// TwinCAT 3 PLC project PLC
// ProgramVersion: 3.1.4023.0
// libraries:
//   JobManagementFramework, * (Bekchoff Automation K.K.)
//   Tc2_EtherCAT, * (Beckhoff Automation GmbH)
//   Tc2_MC2, * (Beckhoff Automation GmbH)
//   Tc2_Standard, * (Beckhoff Automation GmbH)
//   Tc2_System, * (Beckhoff Automation GmbH)
//   Tc2_Utilities, * (Beckhoff Automation GmbH)
//   Tc3_Module, * (Beckhoff Automation GmbH)
//   VisuSymbols,3.5.10.0,System
// project tree:
//   DUTs/ JobEventReport.TcDUT
//   / GlobalTextList.TcGTLO, PlcTask.TcTTO, Visualization Manager.TcVMO (not stored), VISU_TASK.TcTTO
//   POUs/activities/ FB_Observer.TcPOU, FutureMCGearIn.TcPOU, FutureMCGearInCreator.TcPOU (not stored), FutureMCGearOutCreator.TcPOU (not stored), FutureMCGearOut.TcPOU, FutureMCInching.TcPOU, FutureMCInchingCreator.TcPOU (not stored), FutureMCResetCreator.TcPOU (not stored), FutureMCReset.TcPOU (not stored), FutureMCStopCreator.TcPOU (not stored), FutureMCStop.TcPOU, FutureMCMoveVelocityCreator.TcPOU (not stored), FutureMCMoveVelocity.TcPOU, FutureMCMoveRelativeCreator.TcPOU (not stored), FutureMCMoveRelative.TcPOU, FutureMCMoveAbsolute.TcPOU, FutureMCMoveAbsoluteCreator.TcPOU (not stored), FutureSleepCreator.TcPOU (not stored), FutureMCSetPositionCreator.TcPOU (not stored), FutureMCPower.TcPOU, FutureMCHalt.TcPOU, FutureMCPowerCreator.TcPOU, FutureMCHaltCreator.TcPOU (not stored), FutureMCSetPosition.TcPOU, FutureSleep.TcPOU (not stored)
//   POUs/ MAIN.TcPOU
//   VISUs/ Visualization.TcVIS
// real-time tasks:
//   TASK PlcTask: cycle T#1ms, priority 4, ADS port 350
//   TASK VISU_TASK1: cycle T#50000us, priority 30, ADS port 352
// motion (NC):
//   TASK NC-Task 1 SAF: cycle T#2ms, priority 6, ADS port 501
//   TASK NC-Task 1 SVB: cycle T#10ms, priority 10, ADS port 511
//   AXIS Axis 1 (id 1)
//     General: UnitName=Degree
//     Dynamic: AccelerationMaximum=29071, DecelerationMaximum=29071, Acceleration=14535, Deceleration=14535, Jerk=43605
//     Velo: RefSearch=96.9, RefSync=96.9, SlowManual=484.5, FastManual=2907, Fast=9690, Maximum=9690
//     OtherSettings: AllowMotionCmdToSlave=true
//     encoder EncType=19
//       EncPara: ScaleFactorNumerator=360, ScaleFactorDenominator=1048576, MaxCount=#xffffffff
//     drive DrvType=16
//       DrvPara: MaxCount=#xffffffff, DriveControlDWord=#x00020100
//         Analog: VeloReferenz=10659, VeloScale=32, TorqueSetpointScale=10, ScaleFactorActTorque=0.1
//         TimeComp: TaskDelayCycles=1
//     controller CtrType=1
//       CtrPara: PriorControlFactor=1
//         Observer: BandWidth=20
//   AXIS Axis 2 (id 2)
//     General: UnitName=Degree
//     Dynamic: AccelerationMaximum=29071, DecelerationMaximum=29071, Acceleration=14535, Deceleration=14535, Jerk=43605
//     Velo: RefSearch=96.9, RefSync=96.9, FastManual=200, Fast=9690, Maximum=9690
//     OtherSettings: AllowMotionCmdToSlave=true, PulseDistancePos=1, PulseDistanceNeg=1
//     encoder EncType=19
//       EncPara: ScaleFactorNumerator=360, ScaleFactorDenominator=1048576, Inverse=true, MaxCount=#xffffffff
//     drive DrvType=16
//       DrvPara: Inverse=true, MaxCount=#xffffffff, DriveControlDWord=#x00020100
//         Analog: VeloReferenz=10659, VeloScale=32, TorqueSetpointScale=10, ScaleFactorActTorque=0.1
//         TimeComp: TaskDelayCycles=1
//     controller CtrType=1
//       CtrPara: PriorControlFactor=1
//         Observer: BandWidth=20
// I/O:
//   DEVICE Device 2 (EtherCAT), AmsNetId 169.254.89.239.3.1
//     Term 1 (EK1101) [EK1101 EtherCAT Coupler (2A E-Bus, ID switch)]
//       Drive 2 (EL7201-0011) [EL7201-0011 1Ch. DS402 Servo motor output stage with OCT (50V, 4A)]
//       Drive 3 (EL7201-0011) [EL7201-0011 1Ch. DS402 Servo motor output stage with OCT (50V, 2.8A RMS)]
//       Term 4 (EL9011) [EL9011 End Terminal]
// variable links:
//   NC-Task 1 SAF/Axes/Axis 1 <-> Device 2 (EtherCAT)/Term 1 (EK1101)/Drive 2 (EL7201-0011)
//     Drive/Inputs/In/nDataIn1 <-> DS402 Following error actual value/Following error actual value
//     Drive/Inputs/In/nDcOutputTime <-> InfoData/DcOutputShift
//     Drive/Inputs/In/nState1 <-> DS402 Statusword/Statusword
//     Drive/Inputs/In/nState2 <-> DS402 Statusword/Statusword @bit 8
//     Drive/Inputs/In/nState4 @bit 1 <-> WcState/InputToggle
//     Drive/Inputs/In/nState4 <-> WcState/WcState
//     Drive/Outputs/Out/nCtrl1 <-> DS402 Controlword/Controlword
//     Drive/Outputs/Out/nCtrl2 <-> DS402 Controlword/Controlword @bit 8
//     Drive/Outputs/Out/nDataOut1 <-> DS402 Target position/Target position
//     Enc/Inputs/In/nDataIn1 <-> DS402 Position actual value/Position actual value
//     Enc/Inputs/In/nDcInputTime <-> InfoData/DcInputShift
//     Enc/Inputs/In/nState4 @bit 1 <-> WcState/InputToggle
//     Enc/Inputs/In/nState4 <-> WcState/WcState
//   NC-Task 1 SAF/Axes/Axis 2 <-> Device 2 (EtherCAT)/Term 1 (EK1101)/Drive 3 (EL7201-0011)
//     Drive/Inputs/In/nDataIn1 <-> DS402 Following error actual value/Following error actual value
//     Drive/Inputs/In/nDcOutputTime <-> InfoData/DcOutputShift
//     Drive/Inputs/In/nState1 <-> DS402 Statusword/Statusword
//     Drive/Inputs/In/nState2 <-> DS402 Statusword/Statusword @bit 8
//     Drive/Inputs/In/nState4 @bit 1 <-> WcState/InputToggle
//     Drive/Inputs/In/nState4 <-> WcState/WcState
//     Drive/Outputs/Out/nCtrl1 <-> DS402 Controlword/Controlword
//     Drive/Outputs/Out/nCtrl2 <-> DS402 Controlword/Controlword @bit 8
//     Drive/Outputs/Out/nDataOut1 <-> DS402 Target position/Target position
//     Enc/Inputs/In/nDataIn1 <-> DS402 Position actual value/Position actual value
//     Enc/Inputs/In/nDcInputTime <-> InfoData/DcInputShift
//     Enc/Inputs/In/nState4 @bit 1 <-> WcState/InputToggle
//     Enc/Inputs/In/nState4 <-> WcState/WcState
//   PLC/PLC Instance <-> NC-Task 1 SAF/Axes/Axis 1
//     PlcTask Inputs/MAIN.stAxis1.NcToPlc <-> Outputs/ToPlc
//     PlcTask Outputs/MAIN.stAxis1.PlcToNc <-> Inputs/FromPlc
//   PLC/PLC Instance <-> NC-Task 1 SAF/Axes/Axis 2
//     PlcTask Inputs/MAIN.stAxis2.NcToPlc <-> Outputs/ToPlc
//     PlcTask Outputs/MAIN.stAxis2.PlcToNc <-> Inputs/FromPlc

CONFIGURATION PLC
    RESOURCE PLC ON TwinCAT3
        TASK PlcTask(INTERVAL := T#1ms, PRIORITY := 4);
        TASK VISU_TASK(INTERVAL := T#50000us, PRIORITY := 30);
        PROGRAM MAIN WITH PlcTask : MAIN;
        PROGRAM VisuElems_Visu_Prg WITH VISU_TASK : VisuElems.Visu_Prg;
    END_RESOURCE
END_CONFIGURATION

// ---- DUTs/JobEventReport.TcDUT
{attribute 'pack_mode' := '1'}
TYPE JobEventReport :
STRUCT
	{attribute 'TcAnalytics'}
	subject	: STRING(256);
	 {attribute 'TcAnalytics'}
	job_id	: STRING(256);
	 {attribute 'TcAnalytics'}
	old_state	: STRING(16);
	 {attribute 'TcAnalytics'}
	new_state	: STRING(16);
	 {attribute 'TcAnalytics'}
	record_time	: jobmgmt.T_FILETIME64;
END_STRUCT
END_TYPE

// ---- POUs/MAIN.TcPOU
PROGRAM MAIN
VAR
	work_number	: ULINT;
	act_dc_time : T_DCTIME64;
	dc_task_time : T_DCTIME64;
	dc_tick_time : T_DCTIME64;
	diff_time : T_DCTIME64;
	fbConvertDcTimeToPos : ConvertDcTimeToPos;
	position_at_task_start_point : LREAL;
	position_diff : LREAL;
	dc_time_array : ARRAY [0..1] OF T_DCTIME32;

	fbPower1:mc_power;
	fbPower2:mc_power;
	fbJog:MC_Jog;
	basic_job : FB_Executor;
	demo_job : FB_Executor;
	gear_in_job : FB_Executor;
	init_pos_job : FB_Executor;
	jog_plus_job : FB_Executor;
	jog_minus_job : FB_Executor;
	fb_observer : FB_Observer;
	job_reset : BOOL;
	
	mc_power_future_creator: FutureMCPowerCreator;
	mc_reset_future_creator: FutureMCResetCreator;
	mc_set_position_future_creator: FutureMCSetPositionCreator;
	mc_inching_future_creator : FutureMCInchingCreator;
	mc_gear_in_future_creator : FutureMCGearInCreator;
	mc_gear_out_future_creator : FutureMCGearOutCreator;
	mc_move_rel_future_creator : FutureMCMoveRelativeCreator;
	mc_move_abs_future_creator : FutureMCMoveAbsoluteCreator;
	mc_move_velocity_future_creator: FutureMCMoveVelocityCreator;
	mc_stop_future_creator: FutureMCStopCreator;
	sleep_creator : FutureSleepCreator;

	
	iState:INT;
	stAxis1:axis_ref;
	stAxis2:axis_ref;
	bStart: BOOL;
	bJogPlus: BOOL;
	bJogMinus: BOOL;
	bPower: BOOL;
	_bPower : BOOL;
	iPowerState : UINT;
	bReset:BOOL;
	bError:BOOL;
	bAllAxisPowerOn: BOOL;
	bInsync:BOOL;
	create_container: INT;
	boot_up : BOOL := TRUE;
	i: UINT;
	
	quit: INT;
END_VAR


act_dc_time := F_GetActualDcTime64();
dc_task_time := F_GetCurDcTaskTime64();
dc_tick_time := F_GetCurDcTickTime64();

MEMCPY(ADR(dc_time_array), ADR(dc_task_time), SIZEOF(dc_task_time));

fbConvertDcTimeToPos(nAxisId := 1, nSubIdx := 16#10000, dcTime := dc_time_array[0] + 300000);
position_at_task_start_point := fbConvertDcTimeToPos.fPosition;
position_diff := stAxis1.NcToPlc.ActPos - fbConvertDcTimeToPos.fPosition;

diff_time := act_dc_time - dc_task_time;

IF boot_up THEN
	basic_job.create_container(ContainerType.PARALLEL_QUEUE, 'BASIC');
	basic_job.continuous_mode := TRUE;
	basic_job.id := 'M1';
	basic_job.job_event_reporter := fb_observer;
	JobCreate_PosInit(init_pos_job);
	JobCreate_GearIn(gear_in_job);
	JobCreateDemo(demo_job);
	
	

	mc_inching_future_creator.set_parameters(stAxis2, TRUE,1 , 100);
	jog_plus_job.create_future(mc_inching_future_creator,'JOG_PLUS');
	
	mc_inching_future_creator.set_parameters(stAxis2, FALSE, 1, 100);		
	jog_minus_job.create_future(mc_inching_future_creator,'JOG_MINUS');

	boot_up := FALSE;
END_IF


fbPower1(Axis := stAxis1, Enable := bPower, Enable_Positive := TRUE, Enable_Negative := TRUE, Override := 100.0);
fbPower2(Axis := stAxis2, Enable := bPower, Enable_Positive := TRUE, Enable_Negative := TRUE, Override := 100.0);

(*
IF NOT fbPower1.Status AND NOT fbPower2.Status THEN
	IF demo_job.reset(FALSE) THEN
		iState := 0;
	END_IF
END_IF
*)

CASE iState OF
	0:
		IF fbPower1.Status AND fbPower2.Status THEN
			IF init_pos_job.init() THEN
				basic_job.children.append_job(init_pos_job);
				iState := 1;
			END_IF
		END_IF
	1:
		IF init_pos_job.done THEN
			iState := 2;
		END_IF
	2:
		//fbJog(Axis:=stAxis1 , JogForward:=bJogPlus ,JogBackwards:=bJogMinus, Position := 1, Velocity := 100, Mode := E_JogMode.MC_JOGMODE_INCHING );
		IF bJogPlus THEN
			IF jog_plus_job.init() THEN
				basic_job.children.append_job(jog_plus_job);
				bJogPlus := FALSE;				
			END_IF
		END_IF
		
		IF bJogMinus THEN
			IF jog_minus_job.init() THEN
				basic_job.children.append_job(jog_minus_job);
				bJogMinus := FALSE;				
			END_IF
		END_IF

		IF bStart THEN
			IF gear_in_job.init() THEN
				basic_job.children.append_job(gear_in_job);
				iState := 3;
			END_IF
		END_IF
	3:
		IF demo_job.init() THEN
			work_number := work_number + 1;
			demo_job.id := TO_STRING(work_number);
			basic_job.children.append_job(demo_job);
			iState := 4;
		END_IF
	4:
		IF demo_job.done THEN
			IF bStart THEN
				iState := 3;
			ELSE
				iState := 1;
			END_IF
		END_IF
END_CASE


IF bPower THEN
	job_reset := TRUE;
ELSE
	IF job_reset AND basic_job.reset(FALSE) THEN
		iState := 0;
		job_reset := FALSE;
	END_IF
END_IF

basic_job.execute();

bError := basic_job.nErrorID <> 0;

IF bReset THEN
	IF basic_job.error_reset() THEN
		IF basic_job.resume() THEN
			bReset := FALSE;
		END_IF
	END_IF 
END_IF

IF basic_job.ready THEN
	basic_job.start();
END_IF

(*

CASE iState OF
0:
 	IF stAxis1.NcToPlc.ErrorCode = 0 AND  stAxis1.NcToPlc.ErrorCode = 0 THEN
		iState:=20;
	ELSE
		iState:=10;
	END_IF
10:
		fbReset1(Axis:=stAxis1 , Execute:=TRUE , Done=> , Busy=> , Error=> , ErrorID=> );
		fbReset2(Axis:=stAxis2 , Execute:=TRUE , Done=> , Busy=> , Error=> , ErrorID=> );
		IF stAxis1.NcToPlc.ErrorCode = 0 AND  stAxis1.NcToPlc.ErrorCode = 0 THEN
			fbReset1(Axis:=stAxis1 , Execute:=TRUE , Done=> , Busy=> , Error=> , ErrorID=> );
			fbReset2(Axis:=stAxis2 , Execute:=TRUE , Done=> , Busy=> , Error=> , ErrorID=> );
			iState:=20;
		END_IF

20:
   fbPower1(Axis:=stAxis1 , Enable:=bPower ,	Enable_Positive:=bPower , Enable_Negative:=bPower , Override:=100 , BufferMode:= , Options:=  );
   fbPower2(Axis:=stAxis2 , Enable:=bPower ,	Enable_Positive:=bPower , Enable_Negative:=bPower , Override:=100 , BufferMode:= , Options:=  );
	IF fbPower1.Status AND fbPower2.Status AND bPower THEN
		bAllAxisPowerOn:=TRUE;
		iState:=50;
	END_IF
50:
	IF bStart THEN
		iState:=60;
	END_IF
	IF NOT bPower THEN
		iState:=20;
	END_IF
	fbJog(Axis:=stAxis2 , JogForward:=bJogPlus ,JogBackwards:=bJogMinus , );
	
	
60:
   fbSetPosition1(	Axis:=stAxis1 , 	Execute:=TRUE , Position:=0 ,Mode:= , Options:=  );
   fbSetPosition2(	Axis:=stAxis2 , 	Execute:=TRUE , Position:=0 ,Mode:= , Options:=  );
   IF fbSetPosition1.done AND  fbSetPosition2.Done THEN
	   fbSetPosition1(	Axis:=stAxis1 , 	Execute:=FALSE , Position:=0 ,Mode:= , Options:=  );
	   fbSetPosition2(	Axis:=stAxis2 , 	Execute:=FALSE , Position:=0 ,Mode:= , Options:=  );
		iState:=70;	   
   END_IF
70:
	fbGearIn(Master:=stAxis1 ,Slave:=stAxis2 ,Execute:=TRUE ,RatioNumerator:=1 ,RatioDenominator:=1 ,Acceleration:= ,Deceleration:= ,Jerk:= ,BufferMode:= ,	Options:= );
	IF fbGearIn.InGear THEN
		bInsync:=TRUE;
		fbGearIn(Master:=stAxis1 ,Slave:=stAxis2 ,Execute:=FALSE ,RatioNumerator:=1 ,RatioDenominator:=1 ,Acceleration:= ,Deceleration:= ,Jerk:= ,BufferMode:= ,	Options:= );
		iState:=100;
	END_IF
100:
	iMoveCount:=0;
	iMoveCount1:=0;
	lrDiatance:=20;
	iState:=110;
	
110://Demo1
	iState:=120;
120:
    fbMoveRel(Axis:=stAxis1 ,Execute:=TRUE ,Distance:=lrDiatance ,Velocity:=200 );
    IF fbMoveRel.Done THEN
		fbMoveRel(Axis:=stAxis1 ,Execute:=FALSE ,Distance:=lrDiatance ,Velocity:=200 );
		iState:=130;
	END_IF
130:	
   tWaitTimer1(IN:=TRUE,PT:=T#100MS);
   IF tWaitTimer1.Q THEN
	   tWaitTimer1(IN:=FALSE);
		iState:=140;
		iMoveCount:=iMoveCount+1;
   END_IF
140:
	IF iMoveCount > 18 THEN
		iState:=150;
	ELSE
		iState:=110;
     END_IF
150:
    fbMoveAbs1(Axis:=stAxis1 ,	Execute:= TRUE, Position:= 0,Velocity:=700 );	
	IF fbMoveAbs1.Done THEN
		iMoveCount1:=iMoveCount1+1;
		fbMoveAbs1(Axis:=stAxis1 ,	Execute:= FALSE, Position:= 0,Velocity:=700 );
		IF iMoveCount1 > 4 THEN
			iState:=200;
		ELSE
			iMoveCount:=0;
			IF lrDiatance = 20 THEN
				lrDiatance := -20;
			ELSE
				lrDiatance := 20;
			END_IF
			iState:=110;
		END_IF
		
	END_IF
200://Demo2
   tWaitTimer2(IN:=TRUE,PT:=T#100MS);
   IF tWaitTimer2.Q THEN
	   tWaitTimer2(IN:=FALSE);
		iState:=210;
		iMoveCount:=iMoveCount+1;
   END_IF
210:
	fbMoveVelo(	Axis:=stAxis1 ,Execute:=TRUE , Velocity:=1000 ,Direction:=MC_Direction.MC_Positive_Direction );
    IF fbMoveVelo.InVelocity THEN
		fbMoveVelo(	Axis:=stAxis1 ,Execute:=FALSE , Velocity:=1000 ,Direction:=MC_Direction.MC_Positive_Direction );
		iState:=220;
	END_IF
220:
   tWaitTimer3(IN:=TRUE,PT:=T#5S);
   IF tWaitTimer3.Q THEN
	   tWaitTimer3(IN:=FALSE);
		iState:=230;
   END_IF
230:
	fbMoveVelo(	Axis:=stAxis1 ,Execute:=TRUE , Velocity:=500 ,Direction:=MC_Direction.MC_Positive_Direction );
    IF fbMoveVelo.InVelocity THEN
		fbMoveVelo(	Axis:=stAxis1 ,Execute:=FALSE , Velocity:=1000 ,Direction:=MC_Direction.MC_Positive_Direction );
		iState:=240;
	END_IF
240:
   tWaitTimer4(IN:=TRUE,PT:=T#5S);
   IF tWaitTimer4.Q THEN
	   tWaitTimer4(IN:=FALSE);
		iState:=250;
   END_IF
250:
	fbStop(Axis:=stAxis1 , Execute:=TRUE,Deceleration:=100,Jerk:=1000  );
	IF fbStop.Done THEN
		fbStop(Axis:=stAxis1 , Execute:=FALSE  );
		iState:=260;
	END_IF
260:
  tWaitTimer5(IN:=TRUE,PT:=T#3000MS);
   IF tWaitTimer5.Q THEN
	   tWaitTimer5(IN:=FALSE);
		iState:=270;
   END_IF
270:
    fbMoveAbs3(Axis:=stAxis1 ,	Execute:= TRUE, Position:= 0,Velocity:=1000 );	
	tWaitTimer6(IN:=TRUE,PT:=T#5S);
	IF tWaitTimer6.Q THEN
		fbMoveAbs3(Axis:=stAxis1 ,	Execute:= FALSE, Position:= 0,Velocity:=1000 );	
	   tWaitTimer6(IN:=FALSE);
		iState:=280;
	END_IF
	IF fbMoveAbs3.Done THEN
		iState:=300;
		fbMoveAbs3(Axis:=stAxis1 ,	Execute:= FALSE, Position:= 0,Velocity:=1000);
	END_IF
280:
    fbMoveAbs2(Axis:=stAxis1 ,	Execute:= TRUE, Position:= 0,Velocity:=500 );	
	IF fbMoveAbs2.Done THEN
		iState:=1000;
		fbMoveAbs2(Axis:=stAxis1 ,	Execute:= FALSE, Position:= 0,);
	END_IF

	
1000: //End Prodcution Code
	IF NOT bStart THEN
		iState:=1010;
	ELSE
		iState:=100;
	END_IF
1010:
  fbGearOut(Slave:=stAxis2 , Execute:=TRUE );
  IF fbGearOut.Done THEN
		bInsync:=FALSE;
	   fbGearOut(Slave:=stAxis2 , Execute:=FALSE );
		iState:=50;
  END_IF

2000: //error Handle
  fbGearO/.ut(Slave:=stAxis2 , Execute:=TRUE );
  IF fbGearOut.Done THEN
	bInsync:=FALSE;
	fbGearOut(Slave:=stAxis2 , Execute:=FALSE );
	iState:=2010;
  END_IF
2010:
	bPower:=FALSE;
  	fbPower1(Axis:=stAxis1 , Enable:=bPower ,	Enable_Positive:=bPower , Enable_Negative:=bPower , Override:=100 , BufferMode:= , Options:=  );
   	fbPower2(Axis:=stAxis2 , Enable:=bPower ,	Enable_Positive:=bPower , Enable_Negative:=bPower , Override:=100 , BufferMode:= , Options:=  );
	IF NOT fbPower1.Status AND NOT fbPower2.Status THEN
		bAllAxisPowerOn:=FALSE;
		iState:=2020;
	END_IF
2020:
	fbReset1(Axis:=stAxis1 , Execute:= bReset);
	fbReset2(Axis:=stAxis2 , Execute:= bReset);
	bReset:=FALSE;
	IF stAxis1.NcToPlc.ErrorCode = 0 AND stAxis2.NcToPlc.ErrorCode = 0 THEN
		bError:=FALSE;
		fbReset1(Axis:=stAxis1 , Execute:= FALSE);
		fbReset2(Axis:=stAxis2 , Execute:= FALSE);
		iState:=0;
	END_IF 
END_CASE

*)

METHOD Execution : BOOL
VAR_INPUT
	main_job : REFERENCE TO FB_Executor;
	bStart : BOOL := TRUE;
END_VAR
Execution := main_job.execute();

IF main_job.ready THEN
	main_job.start();
END_IF

IF bStart THEN
	main_job.start();
END_IF
END_METHOD

METHOD JobCreate_GearIn : BOOL
VAR_INPUT
	job : REFERENCE TO FB_Executor;
END_VAR
// Gear In
mc_gear_in_future_creator.set_parameters(stAxis1, stAxis2);
job.create_future(mc_gear_in_future_creator,'Gear IN');
END_METHOD

METHOD JobCreate_PosInit : BOOL
VAR_INPUT
	job : REFERENCE TO FB_Executor;
END_VAR
VAR
	_job_temp	: REFERENCE TO FB_Executor; // reference to job object for working.
END_VAR
job.create_container(ContainerType.PARALLEL, 'INIT_POS');
// position set to 0
mc_set_position_future_creator.set_parameters(stAxis1, 0);
_job_temp REF= job.children.create_job(mc_set_position_future_creator,'AXIS1_POS_INIT');

mc_set_position_future_creator.set_parameters(stAxis2, 0);
_job_temp REF= job.children.create_job(mc_set_position_future_creator,'AXIS2_POS_INIT');
END_METHOD

METHOD JobCreateDemo : BOOL
VAR_INPUT
	base_job : REFERENCE TO FB_Executor;
END_VAR
VAR
	_job_temp : REFERENCE TO FB_Executor;
	sleep : POINTER TO FutureSleep;
	sleep_creator : FutureSleepCreator;

	mc_move_rel_future : POINTER TO FutureMCMoveRelative;
	mc_move_rel_future_creator : FutureMCMoveRelativeCreator;

	mc_move_abs_future : POINTER TO FutureMCMoveAbsolute;
	mc_move_abs_future_creator : FutureMCMoveAbsoluteCreator;

	mc_move_velocity_future: POINTER TO FutureMCMoveVelocity;
	mc_move_velocity_future_creator: FutureMCMoveVelocityCreator;

END_VAR
base_job.create_container(ContainerTYpe.BATCH, 'DEMO_JOB');
// Sequence
FOR i := 1 TO 10 DO

	mc_move_rel_future_creator.set_parameters(stAxis1,20,200,0,0,0,0);
	_job_temp REF= base_job.children.create_job(mc_move_rel_future_creator,CONCAT('MOVE20_', TO_STRING(i)));

	sleep_creator.sleep_time := T#100MS;
	_job_temp REF= base_job.children.create_job(sleep_creator,CONCAT('WAIT_100MS_', TO_STRING(i)));
	
END_FOR

// position set to 0

mc_move_abs_future_creator.set_parameters(stAxis1,0,200,0,0,0,0);
_job_temp REF= base_job.children.create_job(mc_move_abs_future_creator,CONCAT('MOVE20_', TO_STRING(i)));

FOR i := 1 TO 10 DO

	mc_move_rel_future_creator.set_parameters(stAxis1,-20,200,0,0,0,0);
	_job_temp REF= base_job.children.create_job(mc_move_rel_future_creator,CONCAT('MOVE-20_', TO_STRING(i)));

	sleep_creator.sleep_time := T#100MS;
	_job_temp REF= base_job.children.create_job(sleep_creator,CONCAT('WAIT_100MS_', TO_STRING(i)));
	
END_FOR

// position to 0

mc_move_abs_future_creator.set_parameters(stAxis1,0,200,0,0,0,0);
_job_temp REF= base_job.children.create_job(mc_move_abs_future_creator,'MOVE_HOME');

sleep_creator.sleep_time := T#100MS;
_job_temp REF= base_job.children.create_job(sleep_creator,'WAIT_100MS');

// 1000deg/s -> 500deg/s

mc_move_velocity_future_creator.set_parameters(stAxis1,MC_Direction.MC_Positive_Direction,1000,0,0,0,0);
_job_temp REF= base_job.children.create_job(mc_move_velocity_future_creator,'VELO-1000');

sleep_creator.sleep_time := T#5S;
_job_temp REF= base_job.children.create_job(sleep_creator,'WAIT_5S');

mc_move_velocity_future_creator.set_parameters(stAxis1,MC_Direction.MC_Positive_Direction,500,0,0,0,0);
_job_temp REF= base_job.children.create_job(mc_move_velocity_future_creator,'VELO-500');

sleep_creator.sleep_time := T#5S;
_job_temp REF= base_job.children.create_job(sleep_creator,'WAIT_5S');

mc_stop_future_creator.set_parameters(stAxis1,0,0);
_job_temp REF= base_job.children.create_job(mc_stop_future_creator,'STOP');

// position to 0

mc_move_abs_future_creator.set_parameters(stAxis1,0,1000,0,0,0,0);
_job_temp REF= base_job.children.create_job(mc_move_abs_future_creator,'MOVE_HOME');
END_METHOD

END_PROGRAM

// ---- POUs/activities/FB_Observer.TcPOU
FUNCTION_BLOCK FB_Observer IMPLEMENTS InterfaceObserver
VAR_INPUT
END_VAR
VAR_OUTPUT
	job_event_report : JobEventReport;
END_VAR
VAR
END_VAR

METHOD subscribe_job_directory : BOOL
VAR_INPUT
	(* Represent reference to subscribed job object*)
	executor	: REFERENCE TO jobmgmt.FB_Executor;
END_VAR
VAR
	job_log : STRING;
END_VAR
job_log := CONCAT(job_log, 'JOB STRUCTURE');
IF executor.future <> 0 THEN
	job_log := CONCAT(job_log, '/ FUTURE_NAME :');
	job_log := CONCAT(job_log, executor.future.future_name);
	job_log := CONCAT(job_log, ',');
END_IF

job_log := CONCAT(job_log, 'JOB_ID');
job_log := CONCAT(job_log, ' : ');
job_log := CONCAT(job_log, executor.uid);

ADSLOGSTR(msgCtrlMask := ADSLOG_MSGTYPE_LOG, msgFmtStr := job_log, strArg := '');
END_METHOD

METHOD subscribe_job_event : BOOL
VAR_INPUT
	(* Subject of event*)
	subject	: T_MaxString;
	(* Job state before transition.*)
	old_state	: jobmgmt.E_FutureExecutionState;
	(* Job state after transition.*)
	new_state	: jobmgmt.E_FutureExecutionState;
	(* File-time at the time of transition.*)
	record_time	: jobmgmt.T_FILETIME64;
	(* Reference to job instance of which transition occurs.*)
	executor	: REFERENCE TO jobmgmt.FB_Executor;
END_VAR
VAR_INST
	fb_timezone_info : FB_GetTimeZoneInformation := (bExecute := TRUE);
END_VAR
VAR
	last_state : STRING;
	current_state : STRING;
	text : T_MaxString;
END_VAR
last_state := TO_STRING(old_state);
current_state := TO_STRING(executor.future.state);

job_event_report.subject := subject;
job_event_report.old_state := TO_STRING(old_state);
job_event_report.new_state := TO_STRING(new_state);
job_event_report.record_time := record_time;
job_event_report.job_id := executor.uid;

fb_timezone_info();
text := FILETIME64_TO_ISO8601(fileTime := record_time, nBias := DINT_TO_INT(fb_timezone_info.tzInfo.bias), bUTC := TRUE,nPrecision := 6);
text := CONCAT(text, '	');
text := CONCAT(text, subject);
text := CONCAT(text, '	');
text := CONCAT(text, current_state);
text := CONCAT(text, '	');
text := CONCAT(text, TO_STRING(executor.nErrorID));
text := CONCAT(text, '	');
text := CONCAT(text, executor.future.future_name);
text := CONCAT(text, '	');
text := CONCAT(text, executor.uid);


ADSLOGSTR(msgCtrlMask := ADSLOG_MSGTYPE_LOG, msgFmtStr := text, strArg := '');

subscribe_job_event := TRUE;
END_METHOD

END_FUNCTION_BLOCK

// ---- POUs/activities/FutureMCPowerCreator.TcPOU
FUNCTION_BLOCK FutureMCPowerCreator IMPLEMENTS InterfaceTaskCreator
VAR_INPUT
END_VAR
VAR_OUTPUT
END_VAR
VAR
	_axis: REFERENCE TO AXIS_REF;
	_override: LREAL := 100.0;
	_enable_positive:	BOOL := TRUE; 
	_enable_negative:	BOOL := TRUE;
	_option : ST_PowerOptions;
	_buffer_mode : MC_BufferMode;
END_VAR

{warning 'add method implementation '}
METHOD create_future : jobmgmt.InterfaceFuture
VAR_INPUT
	(* Specify future name*)
	future_name	: STRING;
END_VAR
VAR
	_p_future : POINTER TO FutureMCPower;
END_VAR
_p_future := __NEW(FutureMCPower);
_p_future^.future_name := future_name;
_p_future^.set_parameters(_axis);
_p_future^.set_options(_enable_positive, _enable_negative, _override, _buffer_mode, _option);
create_future := _p_future^;
END_METHOD

{warning 'add method implementation '}
METHOD destroy_future : jobmgmt.InterfaceFuture
VAR_INPUT
	(* Specify future instance whtat you want to delete.*)
	future	: jobmgmt.InterfaceFuture;
END_VAR
VAR
	_p_future : POINTER TO FutureMCPower;
END_VAR
IF __QUERYPOINTER(future, _p_future) THEN
	__DELETE(_p_future);
	IF _p_future = 0  THEN
		destroy_future := 0;
	END_IF
END_IF
END_METHOD

METHOD set_options : BOOL
VAR_INPUT
	Enable_Positive:	BOOL; 
	Enable_Negative:	BOOL;
	Override:			LREAL := 100;
	buffer_mode : MC_BufferMode;
	option : ST_PowerOptions;
END_VAR
_override := Override;
_enable_positive := Enable_Positive;
_enable_negative := Enable_Negative;
_buffer_mode := buffer_mode;
_option := option;
END_METHOD

METHOD set_parameters : BOOL
VAR_INPUT
	axis : REFERENCE TO AXIS_REF;
END_VAR
_axis REF= axis;
END_METHOD

END_FUNCTION_BLOCK

// ---- POUs/activities/FutureMCPower.TcPOU
{attribute 'enable_dynamic_creation'}
FUNCTION_BLOCK FutureMCPower EXTENDS FB_AbstructFuture
VAR_INPUT
END_VAR
VAR_OUTPUT
END_VAR
VAR
	_axis: REFERENCE TO AXIS_REF;
	_override: LREAL := 100.0;
	_enable_positive:	BOOL := TRUE; 
	_enable_negative:	BOOL := TRUE;
	_fb_power	: MC_Power;
	_mc_reset	: MC_Reset;
	_option : ST_PowerOptions;
	_buffer_mode : MC_BufferMode;
	_error_id :UDINT;
END_VAR

METHOD abort : BOOL // Return TRUE if finish.
_fb_power(
	Axis:= _axis, 
	Enable:= FALSE, 
	Enable_Positive:= FALSE, 
	Enable_Negative:= FALSE, 
	Override:= _override, 
	BufferMode:= _buffer_mode, 
	Options:= _option, 
);	

abort := NOT _fb_power.Status;
END_METHOD

METHOD error_reset : BOOL // Must be overrided if future has any errors.
VAR_INST
	_exec_state : UDINT;
END_VAR
IF _error_id <> 0 THEN
	CASE _exec_state OF
		0:
			_mc_reset(Axis := _axis, Execute := FALSE);
			_mc_reset(Axis:= _axis, Execute := TRUE );
			_exec_state := 1;
		1:
			IF _mc_reset.Busy THEN
				_mc_reset(Axis:= _axis,Execute := FALSE);
			END_IF
	END_CASE
	
	_error_id := _mc_reset.ErrorID;
	error_reset := _mc_reset.Done;
ELSE
	error_reset := TRUE;
END_IF
END_METHOD

METHOD execute : BOOL // Return TRUE if finish.

_fb_power(
	Axis:= _axis, 
	Enable:= TRUE, 
	Enable_Positive:= _enable_positive, 
	Enable_Negative:= _enable_negative, 
	Override:= _override, 
	BufferMode:= _buffer_mode, 
	Options:= _option, 
);

_error_id := _fb_power.ErrorID;
execute := NOT _fb_Power.Status;
END_METHOD

PROPERTY nErrorID : UDINT
GET
nErrorID := _error_id;
END_GET
SET
END_SET
END_PROPERTY

METHOD set_options : BOOL
VAR_INPUT
	Enable_Positive:	BOOL; 
	Enable_Negative:	BOOL;
	Override:			LREAL := 100;
	buffer_mode : MC_BufferMode;
	option : ST_PowerOptions;
END_VAR
_override := Override;
_enable_positive := Enable_Positive;
_enable_negative := Enable_Negative;
_buffer_mode := buffer_mode;
_option := option;
END_METHOD

METHOD set_parameters : BOOL
VAR_INPUT
	axis : REFERENCE TO AXIS_REF;
END_VAR
_axis REF= axis;
END_METHOD

END_FUNCTION_BLOCK

// ---- POUs/activities/FutureMCMoveRelative.TcPOU
{attribute 'enable_dynamic_creation'}
FUNCTION_BLOCK FutureMCMoveRelative EXTENDS FB_AbstructFuture
VAR_INPUT
END_VAR
VAR_OUTPUT
END_VAR
VAR
	_fb_move_rel	: MC_MoveRelative;
	_executor		: FB_Executor;
	_axis: REFERENCE TO AXIS_REF;
	_distance : MC_LREAL;
	_velocity : MC_LREAL;
	_acceleration: MC_LREAL;
	_deceleration: MC_LREAL;
	_jerk		: MC_LREAL;
	_option : ST_MoveOptions;
	_buffer_mode : MC_BufferMode ;
	_error_id :UDINT;
	_exec_state : UDINT;
	_abort_state : UINT;
END_VAR

METHOD abort : BOOL // Return TRUE if finish.
VAR_INST
	future_halt : FutureMcHalt;
END_VAR
CASE _abort_state OF
	0:
		_exec_state := 0;
		future_halt.set_parameters(_axis, _deceleration, _jerk);
		future_halt.future_name := 'HALT MOVE_RELATIVE';
		_executor.future := future_halt;
		_abort_state := 1;
	1:
		IF _executor.execute() AND _executor.nErrorID = 0 THEN
			_abort_state := 2;
		END_IF
		
		IF _executor.current_state = E_FutureExecutionState.wait_for_process THEN
			_executor.start();
		END_IF
	2:
		abort := TRUE;
END_CASE
END_METHOD

METHOD execute : BOOL // Return TRUE if finish.

CASE _exec_state OF
	0:
		_abort_state := 0;
		_fb_move_rel(Axis := _axis,Execute := FALSE);
		_fb_move_rel(
			Execute := TRUE,
			Axis := _axis,
			Distance := _distance,
			Velocity := _velocity,
			Acceleration := _acceleration,
			Deceleration := _deceleration,
			Jerk := _jerk,
			BufferMode := _buffer_mode,
			Options := _option
		);
		_exec_state := 1;
	1:
		IF _fb_move_rel.Busy THEN
			_fb_move_rel(Axis := _axis,Execute := FALSE);
		END_IF
END_CASE

_error_id := _fb_move_rel.ErrorID;
execute := _fb_move_rel.Done OR _fb_move_rel.Error;
END_METHOD

METHOD init : BOOL // Return TRUE if finish.

VAR
	axis: INT;
END_VAR
_exec_state := 0;
_abort_state := 0;
_error_id := _fb_move_rel.ErrorID;
init := TRUE;
END_METHOD

PROPERTY nErrorID : UDINT
GET
nErrorID := _error_id;
END_GET
SET
END_SET
END_PROPERTY

METHOD set_options : BOOL
VAR_INPUT
	option : ST_MoveOptions;
END_VAR
_option := option;
END_METHOD

METHOD set_parameters : BOOL
VAR_INPUT
	axis : REFERENCE TO AXIS_REF;
	distance : MC_LREAL;
	velocity : MC_LREAL;
	acceleration	: MC_LREAL;		// Set deceleration in case let moving axis halt.
	deceleration	: MC_LREAL;		// Set deceleration in case let moving axis halt.
	jerk			: MC_LREAL;		// Set jerk in case let moving axis halt.
	buffer_mode : MC_BufferMode;
END_VAR
_axis REF= axis;
_distance := distance;
_velocity := velocity;
_acceleration := acceleration;
_deceleration := deceleration;
_jerk := jerk;
_buffer_mode := buffer_mode;
END_METHOD

END_FUNCTION_BLOCK

// ---- POUs/activities/FutureMCHalt.TcPOU
{attribute 'enable_dynamic_creation'}
FUNCTION_BLOCK FutureMCHalt EXTENDS FB_AbstructFuture
VAR_INPUT
END_VAR
VAR_OUTPUT
END_VAR
VAR
	_axis: REFERENCE TO AXIS_REF;
	_fb_halt	: MC_Halt;
	_deceleration: MC_LREAL;
	_jerk		: MC_LREAL;
	_option : ST_MoveOptions;
	_buffer_mode : MC_BufferMode;
	_error_id :UDINT;
	_exec_state : UDINT;
END_VAR

METHOD execute : BOOL // Return TRUE if finish.

CASE _exec_state OF
	0:
		_fb_halt(axis := _axis, Execute := FALSE);
		_fb_halt(
			Axis:= _axis,
			Execute := TRUE,
			Jerk := _jerk,
			BufferMode := _buffer_mode,
			Options := _option
		);
		_exec_state := 1;
	1:
		IF _fb_halt.Busy THEN
			_fb_halt(Axis:= _axis,Execute := FALSE);
		END_IF
END_CASE

_error_id := _fb_halt.ErrorID;
execute := _fb_halt.Done OR _fb_halt.Error;
END_METHOD

METHOD init : BOOL // Return TRUE if finish.
_exec_state := 0;
init := TRUE;
END_METHOD

PROPERTY nErrorID : UDINT
GET
nErrorID := _error_id;
END_GET
SET
END_SET
END_PROPERTY

METHOD set_options : BOOL
VAR_INPUT
	buffer_mode : MC_BufferMode;
	option : ST_MoveOptions;
END_VAR
_buffer_mode := buffer_mode;
_option := option;
END_METHOD

METHOD set_parameters : BOOL
VAR_INPUT
	axis : REFERENCE TO AXIS_REF;
	deceleration	: MC_LREAL;		// Set deceleration in case let moving axis halt.
	jerk			: MC_LREAL;		// Set jerk in case let moving axis halt.
END_VAR
_axis REF= axis;
_deceleration := deceleration;
_jerk := jerk;
END_METHOD

END_FUNCTION_BLOCK

// ---- POUs/activities/FutureMCMoveAbsolute.TcPOU
{attribute 'enable_dynamic_creation'}
FUNCTION_BLOCK FutureMCMoveAbsolute EXTENDS FB_AbstructFuture
VAR_INPUT
END_VAR
VAR_OUTPUT
END_VAR
VAR
	_fb_move_abs	: MC_MoveAbsolute;
	_executor		: FB_Executor;
	_axis: REFERENCE TO AXIS_REF;
	_position : MC_LREAL;
	_velocity : MC_LREAL;
	_acceleration: MC_LREAL;
	_deceleration: MC_LREAL;
	_jerk		: MC_LREAL;
	_option : ST_MoveOptions;
	_buffer_mode : MC_BufferMode ;
	_error_id :UDINT;
	_exec_state : UDINT;
	_abort_state : UINT;
END_VAR

METHOD abort : BOOL // Return TRUE if finish.
VAR_INST
	future_halt : FutureMcHalt;
END_VAR
CASE _abort_state OF
	0:
		_exec_state := 0;
		future_halt.set_parameters(_axis, _deceleration, _jerk);
		future_halt.future_name := 'HALT MOVE_RELATIVE';
		_executor.future := future_halt;
		_abort_state := 1;
	1:
		IF _executor.execute() AND _executor.nErrorID = 0 THEN
			_abort_state := 2;
		END_IF
		
		IF _executor.current_state = E_FutureExecutionState.wait_for_process THEN
			_executor.start();
		END_IF
	2:
		abort := TRUE;
END_CASE
END_METHOD

METHOD execute : BOOL // Return TRUE if finish.

CASE _exec_state OF
	0:
		_abort_state := 0;
		_fb_move_abs(Axis := _axis,Execute := FALSE);
		_fb_move_abs(
			Execute := TRUE,
			Axis := _axis,
			Position := _position,
			Velocity := _velocity,
			Acceleration := _acceleration,
			Deceleration := _deceleration,
			Jerk := _jerk,
			BufferMode := _buffer_mode,
			Options := _option
		);
		_exec_state := 1;
	1:
		IF _fb_move_abs.Busy THEN
			_fb_move_abs(Axis := _axis,Execute := FALSE);
		END_IF
END_CASE

_error_id := _fb_move_abs.ErrorID;
execute := _fb_move_abs.Done OR _fb_move_abs.Error;
END_METHOD

METHOD init : BOOL // Return TRUE if finish.

VAR
	axis: INT;
END_VAR
_exec_state := 0;
_abort_state := 0;
_error_id := _fb_move_abs.ErrorID;
init := TRUE;
END_METHOD

PROPERTY nErrorID : UDINT
GET
nErrorID := _error_id;
END_GET
SET
END_SET
END_PROPERTY

METHOD set_options : BOOL
VAR_INPUT
	option : ST_MoveOptions;
END_VAR
_option := option;
END_METHOD

METHOD set_parameters : BOOL
VAR_INPUT
	axis : REFERENCE TO AXIS_REF;
	position : MC_LREAL;
	velocity : MC_LREAL;
	acceleration	: MC_LREAL;		// Set deceleration in case let moving axis halt.
	deceleration	: MC_LREAL;		// Set deceleration in case let moving axis halt.
	jerk			: MC_LREAL;		// Set jerk in case let moving axis halt.
	buffer_mode : MC_BufferMode;
END_VAR
_axis REF= axis;
_position := position;
_velocity := velocity;
_acceleration := acceleration;
_deceleration := deceleration;
_jerk := jerk;
_buffer_mode := buffer_mode;
END_METHOD

END_FUNCTION_BLOCK

// ---- POUs/activities/FutureMCMoveVelocity.TcPOU
{attribute 'enable_dynamic_creation'}
FUNCTION_BLOCK FutureMCMoveVelocity EXTENDS FB_AbstructFuture
VAR_INPUT
END_VAR
VAR_OUTPUT
END_VAR
VAR
	_fb_move_velo	: MC_MoveVelocity;
	_executor		: FB_Executor;
	_axis: REFERENCE TO AXIS_REF;
	_velocity : MC_LREAL;
	_direction : MC_DIRECTION;
	_acceleration: MC_LREAL;
	_deceleration: MC_LREAL;
	_jerk		: MC_LREAL;
	_option : ST_MoveOptions;
	_buffer_mode : MC_BufferMode ;
	_error_id :UDINT;
	_exec_state : UDINT;
	_abort_state : UINT;
END_VAR

METHOD abort : BOOL // Return TRUE if finish.
VAR_INST
	future_halt : FutureMcHalt;
END_VAR
CASE _abort_state OF
	0:
		_exec_state := 0;
		future_halt.set_parameters(_axis, _deceleration, _jerk);
		future_halt.future_name := 'HALT MOVE_RELATIVE';
		_executor.future := future_halt;
		_abort_state := 1;
	1:
		IF _executor.execute() AND _executor.nErrorID = 0 THEN
			_abort_state := 2;
		END_IF
		
		IF _executor.current_state = E_FutureExecutionState.wait_for_process THEN
			_executor.start();
		END_IF
	2:
		abort := TRUE;
END_CASE
END_METHOD

METHOD execute : BOOL // Return TRUE if finish.

CASE _exec_state OF
	0:
		_abort_state := 0;
		_fb_move_velo(Axis := _axis,Execute := FALSE);
		_fb_move_velo(
			Execute := TRUE,
			Axis := _axis,
			Direction := _direction,
			Velocity := _velocity,
			Acceleration := _acceleration,
			Deceleration := _deceleration,
			Jerk := _jerk,
			BufferMode := _buffer_mode,
			Options := _option
		);
		_exec_state := 1;
	1:
		IF _fb_move_velo.Busy THEN
			_fb_move_velo(Axis := _axis,Execute := FALSE);
		END_IF
END_CASE

_error_id := _fb_move_velo.ErrorID;
execute := _fb_move_velo.InVelocity OR _fb_move_velo.Error;
END_METHOD

METHOD init : BOOL // Return TRUE if finish.

VAR
	axis: INT;
END_VAR
_exec_state := 0;
_abort_state := 0;
_error_id := _fb_move_velo.ErrorID;
init := TRUE;
END_METHOD

PROPERTY nErrorID : UDINT
GET
nErrorID := _error_id;
END_GET
SET
END_SET
END_PROPERTY

METHOD set_options : BOOL
VAR_INPUT
	option : ST_MoveOptions;
END_VAR
_option := option;
END_METHOD

METHOD set_parameters : BOOL
VAR_INPUT
	axis : REFERENCE TO AXIS_REF;
	direction : MC_DIRECTION;
	velocity : MC_LREAL;
	acceleration	: MC_LREAL;		// Set deceleration in case let moving axis halt.
	deceleration	: MC_LREAL;		// Set deceleration in case let moving axis halt.
	jerk			: MC_LREAL;		// Set jerk in case let moving axis halt.
	buffer_mode : MC_BufferMode;
END_VAR
_axis REF= axis;
_velocity := velocity;
_direction := direction;
_acceleration := acceleration;
_deceleration := deceleration;
_jerk := jerk;
_buffer_mode := buffer_mode;
END_METHOD

END_FUNCTION_BLOCK

// ---- POUs/activities/FutureMCGearIn.TcPOU
{attribute 'enable_dynamic_creation'}
FUNCTION_BLOCK FutureMCGearIn EXTENDS FB_AbstructFuture
VAR_INPUT
END_VAR
VAR_OUTPUT
END_VAR
VAR
	_fb_gear_in	: MC_GearIn;
	_axis_main: REFERENCE TO AXIS_REF;
	_axis_sub: REFERENCE TO AXIS_REF;
	_ratio_numerator	: MC_LREAL := 1;
	_ratio_denominator	: UINT := 1;
	_acceleration: MC_LREAL;
	_deceleration: MC_LREAL;
	_jerk		: MC_LREAL;
	_option : ST_GearInOptions;
	_buffer_mode : MC_BufferMode;
	_error_id :UDINT;
	_exec_state : UDINT;
END_VAR

METHOD execute : BOOL // Return TRUE if finish.
execute := FALSE;
CASE _exec_state OF
	0:
		_fb_gear_in(Master := _axis_main,Slave := _axis_sub,Execute := FALSE);
		_fb_gear_in(
			Execute := TRUE,
			Master := _axis_main,
			Slave := _axis_sub,
			RatioNumerator := _ratio_numerator,
			RatioDenominator := _ratio_denominator,
			Acceleration := _acceleration,
			Deceleration := _deceleration,
			Jerk := _jerk,
			BufferMode := _buffer_mode,
			Options := _option
		);
		_exec_state := 1;
	1:
		IF _fb_gear_in.Busy THEN
			_fb_gear_in(Master := _axis_main,Slave := _axis_sub,Execute := FALSE);
		END_IF
		IF NOT _fb_gear_in.Execute AND NOT _fb_gear_in.Busy THEN
			_exec_state := 2;
		END_IF
	2:
		IF _fb_gear_in.InGear OR _fb_gear_in.Error THEN
			_exec_state := 3;
		END_IF
	3:
		execute := TRUE;
		
END_CASE

_error_id := _fb_gear_in.ErrorID;
END_METHOD

METHOD init : BOOL // Return TRUE if finish.

VAR
	axis: INT;
END_VAR
_exec_state := 0;
_error_id := _fb_gear_in.ErrorID;
init := TRUE;
END_METHOD

PROPERTY nErrorID : UDINT
GET
nErrorID := _error_id;
END_GET
SET
END_SET
END_PROPERTY

METHOD set_options : BOOL
VAR_INPUT
	ratio_numerator	: MC_LREAL;
	ratio_denominator	: UINT;
	acceleration	: MC_LREAL;		// Set deceleration in case let moving axis halt.
	deceleration	: MC_LREAL;		// Set deceleration in case let moving axis halt.
	jerk			: MC_LREAL;		// Set jerk in case let moving axis halt.
	buffer_mode : MC_BufferMode;
	option : ST_GearInOptions;
END_VAR
_ratio_numerator	:= ratio_numerator;
_ratio_denominator	:= ratio_denominator;
_acceleration := acceleration;
_deceleration := deceleration;
_jerk := jerk;
_buffer_mode := buffer_mode;
_option := option;
END_METHOD

METHOD set_parameters : BOOL
VAR_INPUT
	axis_main : REFERENCE TO AXIS_REF;
	axis_sub : REFERENCE TO AXIS_REF;

END_VAR
_axis_main REF= axis_main;
_axis_sub REF= axis_sub;
END_METHOD

END_FUNCTION_BLOCK

// ---- POUs/activities/FutureMCGearOut.TcPOU
{attribute 'enable_dynamic_creation'}
FUNCTION_BLOCK FutureMCGearOut EXTENDS FB_AbstructFuture
VAR_INPUT
END_VAR
VAR_OUTPUT
END_VAR
VAR
	_fb_gear_out	: MC_GearOut;
	_axis_sub: REFERENCE TO AXIS_REF;
	_ratio_numerator	: MC_LREAL := 1;
	_ratio_denominator	: UINT := 1;
	_option : ST_GearOutOptions;
	_error_id :UDINT;
	_exec_state : UDINT;
END_VAR

METHOD execute : BOOL // Return TRUE if finish.
execute := FALSE;
CASE _exec_state OF
	0:
		_fb_gear_out(Slave := _axis_sub,Execute := FALSE);
		_fb_gear_out(
			Execute := TRUE,
			Slave := _axis_sub,
			Options := _option
		);
		_exec_state := 1;
	1:
		IF _fb_gear_out.Busy THEN
			_fb_gear_out(Slave := _axis_sub,Execute := FALSE);
		END_IF
		IF NOT _fb_gear_out.Execute AND NOT _fb_gear_out.Busy THEN
			_exec_state := 2;
		END_IF
	2:
		IF _fb_gear_out.Done OR _fb_gear_out.Error THEN
			_exec_state := 3;
		END_IF
	3:
		execute := TRUE;
		
END_CASE

_error_id := _fb_gear_out.ErrorID;
END_METHOD

METHOD init : BOOL // Return TRUE if finish.

VAR
	axis: INT;
END_VAR
_exec_state := 0;
_error_id := _fb_gear_out.ErrorID;
init := TRUE;
END_METHOD

PROPERTY nErrorID : UDINT
GET
nErrorID := _error_id;
END_GET
SET
END_SET
END_PROPERTY

METHOD set_options : BOOL
VAR_INPUT
	option : ST_GearOutOptions;
END_VAR
_option := option;
END_METHOD

METHOD set_parameters : BOOL
VAR_INPUT
	axis_sub : REFERENCE TO AXIS_REF;
END_VAR
_axis_sub REF= axis_sub;
END_METHOD

END_FUNCTION_BLOCK

// ---- POUs/activities/FutureMCInching.TcPOU
{attribute 'enable_dynamic_creation'}
FUNCTION_BLOCK FutureMCInching EXTENDS FB_AbstructFuture
VAR_INPUT
END_VAR
VAR_OUTPUT
END_VAR
VAR
	_mc_jog	: MC_Jog;
	_mc_reset	: MC_Reset;
	_abort_executor		: FB_Executor;
	_axis: REFERENCE TO AXIS_REF;
	_direction : BOOL;
	_position : MC_LREAL;
	_velocity : MC_LREAL;
	_acceleration: MC_LREAL;
	_deceleration: MC_LREAL;
	_jerk		: MC_LREAL;
	_mode : E_JogMode ;
	_error_id :UDINT;
	_reset_state : UINT;
END_VAR

METHOD abort : BOOL // Return TRUE if finish.
VAR_INST
	future_halt : FutureMcHalt;
END_VAR
abort := TRUE;
END_METHOD

METHOD error_reset : BOOL // Must be overrided if future has any errors.
VAR_INST
	watch_delay  : TON;
END_VAR
_error_id := _mc_jog.ErrorID;
IF _error_id <> 0 THEN
	CASE _reset_state OF
		0:
			_mc_reset(Axis := _axis, Execute := FALSE);
			_mc_reset(Axis:= _axis, Execute := TRUE );
			watch_delay(IN := FALSE);
			_reset_state := 1;
		1:
			IF _mc_reset.Busy THEN
				_mc_reset(Axis:= _axis,Execute := FALSE);
				_reset_state := 2;
			END_IF
		2:
			IF _error_id = 0 THEN
				error_reset := TRUE;
				_reset_state := 0;
			ELSE
				watch_delay(IN := TRUE, PT := T#1S);
				IF watch_delay.Q THEN
					error_reset := TRUE;
					_reset_state := 0;
				END_IF
			END_IF
	END_CASE
	
	IF _error_id = 0 THEN
		_reset_state := 0;
	END_IF
ELSE
	error_reset := TRUE;
END_IF
END_METHOD

METHOD execute : BOOL // Return TRUE if finish.
_mc_jog(
	JogForward := _direction,
	JogBackwards := NOT _direction,
	Axis := _axis,
	Position := _position,
	Velocity := _velocity,
	Acceleration := _acceleration,
	Deceleration := _deceleration,
	Jerk := _jerk,
	Mode := E_JogMode.MC_JOGMODE_INCHING
);

_error_id := _mc_jog.ErrorID;
execute := _mc_jog.Done OR _mc_jog.Error;
END_METHOD

METHOD init : BOOL // Return TRUE if finish.

VAR
	axis: INT;
END_VAR
_reset_state := 0;
_error_id := _mc_jog.ErrorID;
init := TRUE;
END_METHOD

PROPERTY nErrorID : UDINT
GET
nErrorID := _error_id;
END_GET
SET
END_SET
END_PROPERTY

METHOD set_options : BOOL
VAR_INPUT
	acceleration	: MC_LREAL;		// Set deceleration in case let moving axis halt.
	deceleration	: MC_LREAL;		// Set deceleration in case let moving axis halt.
	jerk			: MC_LREAL;		// Set jerk in case let moving axis halt.
END_VAR
_acceleration := acceleration;
_deceleration := deceleration;
_jerk := jerk;
END_METHOD

METHOD set_parameters : BOOL
VAR_INPUT
	axis : REFERENCE TO AXIS_REF;
	direction : BOOL;
	position : MC_LREAL;
	velocity : MC_LREAL;
END_VAR
_axis REF= axis;
_direction := direction;
_position := position;
_velocity := velocity;
END_METHOD

END_FUNCTION_BLOCK

// ---- POUs/activities/FutureMCStop.TcPOU
{attribute 'enable_dynamic_creation'}
FUNCTION_BLOCK FutureMCStop EXTENDS FB_AbstructFuture
VAR_INPUT
END_VAR
VAR_OUTPUT
END_VAR
VAR
	_axis: REFERENCE TO AXIS_REF;
	_mc_stop	: MC_Stop;
	_deceleration: MC_LREAL;
	_jerk		: MC_LREAL;
	_option : ST_MoveOptions;
	_error_id :UDINT;
	_exec_state : UDINT;
END_VAR

METHOD execute : BOOL // Return TRUE if finish.

CASE _exec_state OF
	0:
		_mc_stop(axis := _axis, Execute := FALSE);
		_mc_stop(
			Axis:= _axis,
			Execute := TRUE,
			Jerk := _jerk,
			Options := _option
		);
		_exec_state := 1;
	1:
		IF _mc_stop.Busy THEN
			_mc_stop(Axis:= _axis,Execute := FALSE);
		END_IF
END_CASE

_error_id := _mc_stop.ErrorID;
execute := _mc_stop.Done OR _mc_stop.Error;
END_METHOD

METHOD init : BOOL // Return TRUE if finish.
_exec_state := 0;
init := TRUE;
END_METHOD

PROPERTY nErrorID : UDINT
GET
nErrorID := _error_id;
END_GET
SET
END_SET
END_PROPERTY

METHOD set_options : BOOL
VAR_INPUT
	option : ST_MoveOptions;
END_VAR
_option := option;
END_METHOD

METHOD set_parameters : BOOL
VAR_INPUT
	axis : REFERENCE TO AXIS_REF;
	deceleration	: MC_LREAL;		// Set deceleration in case let moving axis halt.
	jerk			: MC_LREAL;		// Set jerk in case let moving axis halt.
END_VAR
_axis REF= axis;
_deceleration := deceleration;
_jerk := jerk;
END_METHOD

END_FUNCTION_BLOCK

// ---- POUs/activities/FutureMCSetPosition.TcPOU
{attribute 'enable_dynamic_creation'}
FUNCTION_BLOCK FutureMCSetPosition EXTENDS FB_AbstructFuture
VAR_INPUT
END_VAR
VAR_OUTPUT
END_VAR
VAR
	_fb_set_position	: MC_SetPosition;
	_axis: REFERENCE TO AXIS_REF;
	_position	: MC_LREAL;
	_mode		: BOOL;
	_option 	: ST_SetPositionOptions;
	_error_id :UDINT;
	_exec_state : UDINT;
END_VAR

METHOD abort : BOOL // Return TRUE if finish.
END_METHOD

METHOD execute : BOOL // Return TRUE if finish.

CASE _exec_state OF
	0:
		_fb_set_position( Axis:= _axis, Execute := FALSE);
		_fb_set_position(
				Axis := _axis,
				Execute := TRUE, 
				Position := _position,
				Mode := _mode,
				Options := _option
		);
		_exec_state := 1;
	1:
		IF _fb_set_position.Busy THEN
			_fb_set_position( Axis:= _axis, Execute := FALSE);
		END_IF
END_CASE

_error_id := _fb_set_position.ErrorID;
execute := _fb_set_position.Done OR _fb_set_position.Error;
END_METHOD

METHOD init : BOOL // Return TRUE if finish.
_exec_state := 0;
init := TRUE;
END_METHOD

PROPERTY nErrorID : UDINT
GET
nErrorID := _error_id;
END_GET
SET
END_SET
END_PROPERTY

METHOD set_options : BOOL
VAR_INPUT
	mode		: BOOL;
	option 	: ST_SetPositionOptions;
END_VAR
_mode := mode;
_option := option;
END_METHOD

METHOD set_parameters : BOOL
VAR_INPUT
	axis: REFERENCE TO AXIS_REF;
	position	: MC_LREAL;
END_VAR
_axis REF= axis;
_position := position;
END_METHOD

END_FUNCTION_BLOCK

// ---- GlobalTextList.TcGTLO
TEXTLIST GlobalTextList
  812 = '%3.1f'
  594 = '%s'
  349 = 'Axis 1-2'
  598 = 'Axis 1-2\nCoupled'
  123 = 'Axis1'
  443 = 'Axis2'
  713 = 'Coupled'
  774 = 'JOB ID'
  873 = 'Jog+'
  237 = 'Jog-'
  351 = 'Power'
  839 = 'PROCESS'
  624 = 'Process'
  832 = 'Reset'
  712 = 'Start'
  645 = 'Time (UTC)'
  776 = '電子ギアON'
END_TEXTLIST

// ---- VISUs/Visualization.TcVIS
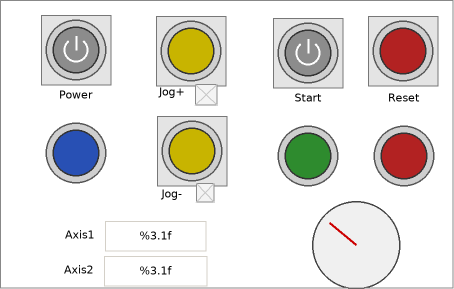
VISUALIZATION Visualization  // 454x289
    Lamp1 (41,118 70x70), variable: MAIN.bAllAxisPowerOn, style: Lamp-Lamp1-Blue
    PowerSwitch (41,15 70x70), variable: MAIN.bPower, behaviour: TOGGLE, style: Switch-PowerSwitch-Gray
    Label (26,80 100x30), "Power"
    PushSwitch (156,16 70x70), variable: MAIN.bJogPlus, behaviour: TOGGLE, style: Switch-PushSwitch-Yellow
    Label (122,77 100x30), "Jog+"
    Label (122,179 100x30), "Jog-"
    PushSwitch (157,116 70x70), variable: MAIN.bJogMinus, behaviour: TOGGLE, style: Switch-PushSwitch-Yellow
    PowerSwitch (273,18 70x70), variable: MAIN.bStart, behaviour: TOGGLE, style: Switch-PowerSwitch-Gray
    Lamp1 (273,121 70x70), variable: MAIN.bStart, style: Lamp-Lamp1-Green
    Label (258,83 100x30), "Start"
    Lamp1 (369,121 70x70), variable: MAIN.bError, style: Lamp-Lamp1-Red
    Label (354,83 100x30), "Reset"
    PushSwitch (368,16 70x70), variable: MAIN.bReset, behaviour: TOGGLE, style: Switch-PushSwitch-Red
    Textfield (105,221 101x30), "%3.1f", text variable: MAIN.stAxis1.NcToPlc.ActPos
    Label (47,220 66x30), "Axis1"
    Label (46,255 66x30), "Axis2"
    Textfield (104,256 103x30), "%3.1f", text variable: MAIN.stAxis2.NcToPlc.ActPos
    Image (195,84 22x21), image: VisuSymbols.Symbols.ArrowHalfLeftLeft
    Image (196,183 18x19), image: VisuSymbols.Symbols.ArrowHalfRightDown
    Meter180 (259,201 194x88), value: MAIN.stAxis1.NcToPlc.ActVelo, style: Meter-Meter180-Blue, scale format: %.1f, scale -1000..1000
END_VISUALIZATION
